FUNCTION_BLOCK F_MUX_2_2
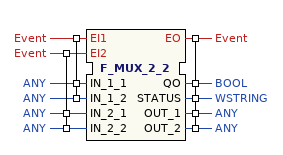
  EVENT_INPUT
    EI1 WITH IN_1_1, IN_1_2;
    EI2 WITH IN_2_1, IN_2_2;
  END_EVENT
  EVENT_OUTPUT
    EO WITH QO, STATUS, OUT_1, OUT_2;
  END_EVENT
  VAR_INPUT
    IN_1_1 : ANY;
    IN_1_2 : ANY;
    IN_2_1 : ANY;
    IN_2_2 : ANY;
  END_VAR
  VAR_OUTPUT
    QO : BOOL;
    STATUS : WSTRING;
    OUT_1 : ANY;
    OUT_2 : ANY;
  END_VAR
END_FUNCTION_BLOCK
